PROGRAM P_Invoke
VAR
	fbInvoke : FB_Invokable;
END_VAR

{attribute 'TcRpcEnable'}
METHOD Meth : INT
VAR_INPUT
	Value : INT;
END_VAR
Meth := Value*2;
END_METHOD

END_PROGRAM

(* stored: Version 1.1.0.1
   POU P_Invoke: Id {186187b0-d27d-4c73-ad36-5d0ff2124d6a}, SpecialFunc None
   Method Meth: Id {d6bac87f-ee1a-4924-bdf7-1aac2b686ad8} *)
